// TIA Portal V20 export
FUNCTION_BLOCK "FB_Vacuums"   // FB441, SCL
{ S7_Optimized_Access := 'TRUE' }
// stored: AutoNumber false, MemoryReserve 100, SetENOAutomatically false
   VAR
      sOutVacuum1On : Bool;
      sControlVacuum1 { S7_SetPoint := 'True'} : "FB_AnalogInputThreshold";
      sCtrlPressureVacuum1 { S7_SetPoint := 'True'} : "FB_AnalogInputThreshold";
      sAspirationLeft { S7_SetPoint := 'True'} : "FB_AnalogInputThreshold";
      sAspirationRight { S7_SetPoint := 'True'} : "FB_AnalogInputThreshold";
      sRT_AspirationKeys { S7_SetPoint := 'True'} : R_TRIG;
      sFT_AspirationKeys { S7_SetPoint := 'True'} : F_TRIG;
      sAspirationKeys { S7_SetPoint := 'True'} : Bool;
   END_VAR
BEGIN
   REGION Description header 
       //==================================================================================
       // POSALUX Swiss SA / (C) Copyright 2024
       //----------------------------------------------------------------------------------
       // Title: Vacuums management
       // Comment/Function: This function manages the machine's suction system, controlling
       //                   six suction circuits.
       // Author: Gowsigan SRITHARAN
       // Engineering: TIA Portal v17
       //----------------------------------------------------------------------------------
       // Change log table:
       // Version  | Date     | Expert in charge | Changes applied
       // ---------|----------|------------------|------------------------------------
       // 00.00.01 | 20241120 | GSR              | First released version
       // ---------|----------|------------------|------------------------------------
       // 00.00.02 | 20250327 | WFA              | Management of only one vacuum
       // ==================================================================================
   END_REGION

   REGION Elbaron vacuum
       // Deactivation of the MCP button (MCP Keyboard 9) in Auto mode
       "DB_McpKeyboardSignals".sK9_Aspiration.sKeyDisable := "LBP_ModeGroup".E_AUTO OR "DB_GestionWorkingModes".sMCP_KxxKeysDisable;
       "DB_HmiKeyboardSignals".sK9_Aspiration.sKeyDisable := "LBP_ModeGroup".E_AUTO;

       #sRT_AspirationKeys(CLK := "DB_McpKeyboardSignals".sK9_Aspiration.sKeySWTogglePositiveFront
                           OR "DB_HmiKeyboardSignals".sK9_Aspiration.sKeySWTogglePositiveFront);

       #sFT_AspirationKeys(CLK := "DB_McpKeyboardSignals".sK9_Aspiration.sKeySWToggleNegativeFront
                           OR "DB_HmiKeyboardSignals".sK9_Aspiration.sKeySWToggleNegativeFront);

       IF #sRT_AspirationKeys.Q THEN
           #sAspirationKeys := TRUE;
       ELSIF #sFT_AspirationKeys.Q THEN
           #sAspirationKeys := FALSE;
       END_IF;

       // Activation of the Elbaron output
       "DB_DigitalOutputs".sElbaronPowerON.sSWStatus :=
       "DB_PowerOn".sMachineReadySoft
       AND NOT "DB_Machineshutdown_UPS".sShutDownAspiration
       AND ((("LBP_Chan1".E_ProgRunning
       OR "LBP_Chan1".E_ProgWait
       OR "LBP_Chan1".E_ProgStop
       OR "LBP_Chan2".E_ProgRunning
       OR "LBP_Chan2".E_ProgWait
       OR "LBP_Chan2".E_ProgStop)
       AND "LBP_ModeGroup".E_AUTO)
       OR #sAspirationKeys);

       // Keys Elbaron Aspiration
       "DB_McpKeyboardSignals".sK9_Aspiration.sKeySWToggleStatus := "DB_DigitalOutputs".sElbaronPowerON.sSWStatus;
       "DB_HmiKeyboardSignals".sK9_Aspiration.sKeySWToggleStatus := "DB_DigitalOutputs".sElbaronPowerON.sSWStatus;

       // LED Elbaron Aspiration
       "DB_McpKeyboardSignals".sK9_Aspiration.sLedSWStatus := "DB_DigitalOutputs".sElbaronPowerON.sSWStatus;
       "DB_HmiKeyboardSignals".sK9_Aspiration.sLedSWStatus := "DB_DigitalOutputs".sElbaronPowerON.sSWStatus;
   END_REGION

   REGION Aspirations control
       #sAspirationLeft(iActualValue := "DB_AnalogInputs".sLeftAspiration.sSWRealValue,
                        iStartDelay := "DB_DigitalOutputs".sElbaronPowerON.sSWStatus,
                        ioAlarmMin := "LBP_AlarmMsgs".UserA[06].A70UUxx[56],
                        ioWarningMin := "LBP_AlarmMsgs".UserA[07].A70UUxx[56],
                        ioWarningMax := "LBP_AlarmMsgs".UserA[07].A70UUxx[57],
                        ioAlarmMax := "LBP_AlarmMsgs".UserA[06].A70UUxx[57],
                        oDataAction => "DB_AnalogInputAction".Left_Aspiration,
                        iDataPLC := "DB_AnalogInputDataPLC".Left_Aspiration,
                        iDataHMI := "DB_AnalogInputDataHMI".Left_Aspiration);

       #sAspirationRight(iActualValue := "DB_AnalogInputs".sRightAspiration.sSWRealValue,
                         iStartDelay := "DB_DigitalOutputs".sElbaronPowerON.sSWStatus,
                         ioAlarmMin := "LBP_AlarmMsgs".UserA[06].A70UUxx[58],
                         ioWarningMin := "LBP_AlarmMsgs".UserA[07].A70UUxx[58],
                         ioWarningMax := "LBP_AlarmMsgs".UserA[07].A70UUxx[59],
                         ioAlarmMax := "LBP_AlarmMsgs".UserA[06].A70UUxx[59],
                         oDataAction => "DB_AnalogInputAction".Right_Aspiration,
                         iDataPLC := "DB_AnalogInputDataPLC".Right_Aspiration,
                         iDataHMI := "DB_AnalogInputDataHMI".Right_Aspiration);
   END_REGION
END_FUNCTION_BLOCK
